DATA_BLOCK "dbEquipTank"
{ S7_Optimized_Access := 'TRUE' }
VERSION : 0.8
NON_RETAIN
   VAR
      equipmentTank { ExternalWritable := 'False'} : Array[1..25] of "tEquipment";
      ia { ExternalAccessible := 'False'; ExternalVisible := 'False'; ExternalWritable := 'False'} : "tIndex";
      firstRunning { ExternalAccessible := 'False'; ExternalVisible := 'False'; ExternalWritable := 'False'} : "tStatus";
   END_VAR


BEGIN

END_DATA_BLOCK

